FUNCTION_BLOCK FB_TriggerManager IMPLEMENTS I_TriggerManager
VAR
    nEL1252LatchPos AT %I* : ULINT;
    nEL1252LatchPosPreviousCycle : ULINT;
    bNewLatchPending : BOOL;
END_VAR


IF nEL1252LatchPos <> nEL1252LatchPosPreviousCycle THEN
    bNewLatchPending := TRUE;
END_IF
nEL1252LatchPosPreviousCycle := nEL1252LatchPos;

{warning 'Add method implementation '}
METHOD GetAndResetTrigger
VAR_OUTPUT
    bLatchDetected	: BOOL;
    (* [ns]*)
    nLatchTime_ns	: ULINT;
END_VAR

bLatchDetected := bNewLatchPending;

nLatchTime_ns := nEL1252LatchPos;

bNewLatchPending := FALSE;
END_METHOD

END_FUNCTION_BLOCK

(* stored: Version 1.1.0.1
   POU FB_TriggerManager: Id {6f90d946-2f37-4b1a-93b8-148c912aa4e6}, SpecialFunc None
   Method GetAndResetTrigger: Id {19ec8f4e-eec6-4c53-8172-d0a6638ebf65} *)
